SYSTEM PNP_VIEWL (* Pick & Place View Tester *)
  (* Standard: IEC 61499; Classification: Simulation; ApplicationDomain: Assembly; Type: Pick & Place *)
  (* Version 0.0, 2006-06-21, JHC, Holobloc Inc, Adapted from ASM_VIEWL *)
  DEVICE HMI : FRAME_DEVICE(BOUNDS := [100,100,325,125], GRID := [3,1])
    RESOURCE CONVEYOR : PANEL_RESOURCE
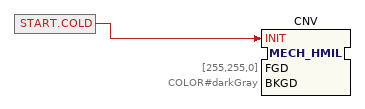
      FBS
        CNV : MECH_HMIL(FGD := [255,255,0], BKGD := COLOR#darkGray);
      END_FBS
      EVENT_CONNECTIONS
        START.COLD TO CNV.INIT;
      END_CONNECTIONS
    END_RESOURCE
    RESOURCE PNP : PANEL_RESOURCE
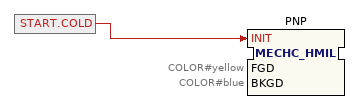
      FBS
        PNP : MECHC_HMIL(FGD := COLOR#yellow, BKGD := COLOR#blue);
      END_FBS
      EVENT_CONNECTIONS
        START.COLD TO PNP.INIT;
      END_CONNECTIONS
    END_RESOURCE
    RESOURCE FAULT : PANEL_RESOURCE
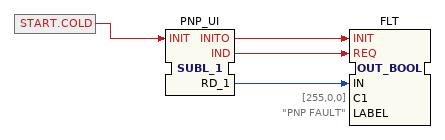
      FBS
        PNP_UI : SUBL_1;
        FLT : OUT_BOOL(C1 := [255,0,0], LABEL := "PNP FAULT");
      END_FBS
      EVENT_CONNECTIONS
        START.COLD TO PNP_UI.INIT;
        PNP_UI.INITO TO FLT.INIT;
        PNP_UI.IND TO FLT.REQ;
      END_CONNECTIONS
      DATA_CONNECTIONS
        PNP_UI.RD_1 TO FLT.IN;
      END_CONNECTIONS
    END_RESOURCE
  END_DEVICE
  DEVICE VIEW : FRAME_DEVICE(BOUNDS := [425,100,160,180])
    RESOURCE PNP : VIEW_PANEL(DIA := 25, SIZE := [6,5], VERTICAL := 0)
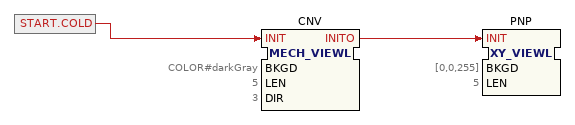
      FBS
        PNP : XY_VIEWL(BKGD := [0,0,255], LEN := 5);
        CNV : MECH_VIEWL(BKGD := COLOR#darkGray, LEN := 5, DIR := 3); (* Conveyor *)
      END_FBS
      EVENT_CONNECTIONS
        START.COLD TO CNV.INIT;
        CNV.INITO TO PNP.INIT;
      END_CONNECTIONS
    END_RESOURCE
  END_DEVICE
END_SYSTEM
